SYSTEM System
  DEVICE M251 : M251_dPAC
    RESOURCE RES0 : EMB_RES_ECO
      FBS
        M251_HSCAction : hscAction;
        FB1 : SYMLINKMULTIVARSRC_1559B0FF8170C9BA0(QI := TRUE, NAME1 := '$${PATH}FEn', VALUE1 := TRUE); {SET_ATTRIBUTE(Configuration.GenericFBType.InterfaceParams, Runtime.System#I:=1;VALUE${I$}:BOOL)}
        FB2 : DPAC_FULLINIT;
        FB3 : EVENTCHAINHEAD(NAME := 'INIT');
        extender_test : TWO_POS_AXIS;
        conveyor_transport : TWO_POS_CONVEYOR_TRANSPORT;
        conveyor_counter : CONVEYOR_WITH_COUNTER;
        shared_compressor : SHARED_COMPRESSOR;
        encoder_axis : ENCODER_AXIS_SINGLE_PHASE;
        vacuum_control : VACUUM_CONTROL;
        BMTM3 : BMTM3(busId := 'BMTM3', enableSymlinkOC := TRUE, phase := T#0ms, busCycleTime := T#5ms, busCycleTolerance := 30, busCycleActionWhenMissed := 1);
        TM251MDESE : TM251MDESE;
        TM3XHSC202_G : TM3XHSC202_G;
        WH_Counter_Hor : HSC_Simple(HscAction := '', CurrentValue := '', ModuloFlag := '', Valid := '', Run := '', ErrorId := '', InstanceName := 'WH_Counter_Hor', ScanRate := 100);
        WH_Counter_Vert : HSC_Simple(HscAction := '', CurrentValue := '', ModuloFlag := '', Valid := '', Run := '', ErrorId := '', InstanceName := 'WH_Counter_Vert', ScanRate := 100);
        ROB_Counter_Vert : HSC_Simple(HscAction := '', CurrentValue := '', ModuloFlag := '', Valid := '', Run := '', ErrorId := '', InstanceName := 'ROB_Counter_Vert', ScanRate := 100);
        ROB_Counter_Hor : HSC_Simple(HscAction := '', CurrentValue := '', ModuloFlag := '', Valid := '', Run := '', ErrorId := '', InstanceName := 'ROB_Counter_Hor', ScanRate := 100);
        ROB_Counter_Rot : HSC_Simple(HscAction := '', CurrentValue := '', ModuloFlag := '', Valid := '', Run := '', ErrorId := '', InstanceName := 'ROB_Counter_Rot', ScanRate := 100);
        TM3DI16_G : TM3DI16_G(DI00 := 'encoder_axis.SensorDriver.ref_switch', DI01 := 'conveyor_transport.sensor2', DI02 := 'conveyor_transport.sensor1', DI03 := '', DI04 := '', DI05 := '', DI06 := 'extender_test.extended_ref_switch', DI07 := 'extender_test.retracted_ref_switch', DI08 := '', DI09 := '', DI10 := '', DI11 := '', DI12 := '', DI13 := '', DI14 := '', DI15 := '');
        TM3DI16_G_1 : TM3DI16_G(DI00 := '', DI01 := '', DI02 := '', DI03 := '', DI04 := '', DI05 := '', DI06 := '', DI07 := '', DI08 := '', DI09 := '', DI10 := '', DI11 := '', DI12 := '', DI13 := '', DI14 := '', DI15 := '');
        TM3AM6_G : TM3AM6_G(AI00 := '', AI01 := '', AI02 := '', AI03 := '', AO00 := '', AO01 := '', AO00_Status := '', AO01_Status := '');
        TM3DQ16T_G : TM3DQ16T_G(DO00 := '', DO01 := '', DO02 := '', DO03 := '', DO04 := '', DO05 := '', DO06 := '', DO07 := '', DO08 := '', DO09 := '', DO10 := '', DO11 := '', DO12 := '', DO13 := '', DO14 := '', DO15 := '');
        TM3DQ32TK : TM3DQ32TK(DO00 := '', DO01 := '', DO02 := '', DO03 := '', DO04 := '', DO05 := '', DO06 := '', DO07 := '', DO08 := '', DO09 := '', DO10 := '', DO11 := '', DO12 := '', DO13 := '', DO14 := '', DO15 := '', DO16 := '', DO17 := '', DO18 := '', DO19 := '', DO20 := '', DO21 := '', DO22 := '', DO23 := '', DO24 := '', DO25 := '', DO26 := '', DO27 := '', DO28 := '', DO29 := '', DO30 := '', DO31 := '');
      END_FBS
      EVENT_CONNECTIONS
        M251_HSCAction.INITO TO FB1.INIT;
        START.COLD TO FB2.INIT;
        START.WARM TO FB2.INIT;
        START.ONLINECHANGE TO FB2.INIT;
        FB2.INITO TO M251_HSCAction.INIT;
        FB1.INITO TO FB3.INIT;
        FB3.INITO TO FB3.TRIGGER;
      END_CONNECTIONS
      ADAPTER_CONNECTIONS
        BMTM3.BusOut TO TM251MDESE.BusIn;
        TM251MDESE.BusOut TO TM3XHSC202_G.BusIn;
        TM3XHSC202_G.IHscChannelOut TO WH_Counter_Hor.IHscChannelIn;
        WH_Counter_Hor.IHscChannelOut TO WH_Counter_Vert.IHscChannelIn;
        WH_Counter_Vert.IHscChannelOut TO ROB_Counter_Vert.IHscChannelIn;
        ROB_Counter_Vert.IHscChannelOut TO ROB_Counter_Hor.IHscChannelIn;
        ROB_Counter_Hor.IHscChannelOut TO ROB_Counter_Rot.IHscChannelIn;
        TM3XHSC202_G.BusOut TO TM3DI16_G.BusIn;
        TM3DI16_G.BusOut TO TM3DI16_G_1.BusIn;
        TM3DI16_G_1.BusOut TO TM3AM6_G.BusIn;
        TM3AM6_G.BusOut TO TM3DQ16T_G.BusIn;
        TM3DQ16T_G.BusOut TO TM3DQ32TK.BusIn;
      END_CONNECTIONS
    END_RESOURCE
  END_DEVICE
END_SYSTEM
